PROGRAM Pneumatic_Axis
VAR
    fbPneumaticAxis : FB_PNEUMATIC_AXIS;

END_VAR

fbPneumaticAxis();
fbPneumaticAxis.stPneumaticAxisInputs.bPermit := TRUE;

END_PROGRAM

(* stored: Version 1.1.0.1, ProductVersion 3.1.4024.5
   POU Pneumatic_Axis: Id {c5a87a8f-b672-49f9-9218-441b3e670d3f}, SpecialFunc None *)
